FUNCTION_BLOCK PID (* Composite Function Block Type *)
  (* Standard: 61499-2 *)
  (* Version 1.0.1, 10/18/2023, ApplicationLibDevTeam, Schneider Electric, First Version *)
  PACKAGE Main;
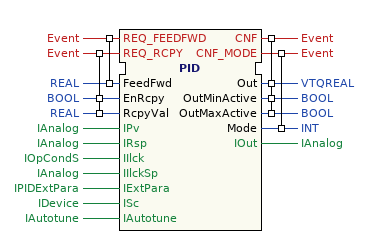
  EVENT_INPUT
    REQ_FEEDFWD WITH FeedFwd; (* Request for executing feedforward gain *)
    REQ_RCPY WITH EnRcpy, RcpyVal; (* Request for actuator position *)
  END_EVENT
  EVENT_OUTPUT
    CNF WITH Out, OutMinActive, OutMaxActive; (* Cyclic execution confirmation *)
    CNF_MODE WITH Mode; (* Execution of confirmation current setpoint *)
  END_EVENT
  VAR_INPUT
    FeedFwd : REAL; (* Feed forward value *)
    EnRcpy : BOOL; (* 1 = the RCPY is enabled *)
    RcpyVal : REAL; (* RCPY value (actuator position) *)
  END_VAR
  VAR_OUTPUT
    Out : VTQREAL; (* Calculated output value *)
    OutMinActive : BOOL; (* 1 = Out has reached OutMin Limit *)
    OutMaxActive : BOOL; (* 1 = Out has reached OutMax Limit *)
    Mode : INT; (* Current mode selected for PID calculation *)
  END_VAR
  SOCKETS
    IPv : IAnalog; (* Process value (range considered) interface adapter *)
    IRsp : IAnalog; (* Program remote setpoint interface adapter *)
    IIlck : IOpCondS; (* Interlock condition summary chain input from ilckCondItem blocks *)
    IIlckSp : IAnalog; (* Interlock setpoint interface adapter, Setpoint to be considered if interlock condition is active *)
    IExtPara : IPIDExtPara; (* External PID parameters interface adapter *)
    ISc : IDevice; (* Sequence control adapter, Controls the block when owner is in program local *)
    IAutotune : IAutotune;
  END_SOCKETS
  PLUGS
    IOut : IAnalog; (* Current output status Interface adapter *)
  END_PLUGS
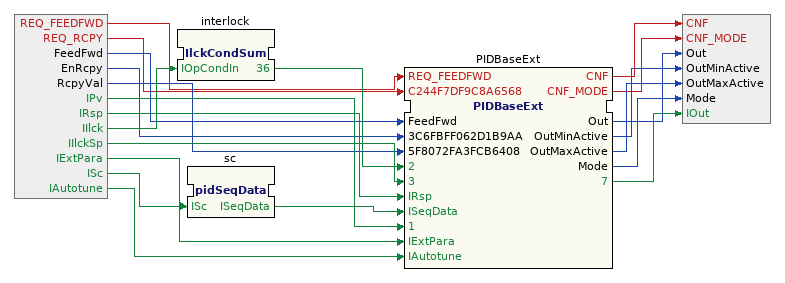
  (* PID Control *)
  (* Interlock *)
  (* Sequence Control *)
  FBS
    interlock : IlckCondSum; {SET_ATTRIBUTE(Configuration.Component.HideUnusedPorts, )}
    sc : pidSeqData;
    PIDBaseExt : PIDBaseExt;
  END_FBS
  EVENT_CONNECTIONS
    REQ_FEEDFWD TO PIDBaseExt.REQ_FEEDFWD;
    PIDBaseExt.CNF TO CNF;
    PIDBaseExt.CNF_MODE TO CNF_MODE;
    REQ_RCPY TO PIDBaseExt.C244F7DF9C8A6568;
  END_CONNECTIONS
  DATA_CONNECTIONS
    FeedFwd TO PIDBaseExt.FeedFwd;
    PIDBaseExt.Out TO Out;
    PIDBaseExt.OutMinActive TO OutMinActive;
    PIDBaseExt.OutMaxActive TO OutMaxActive;
    PIDBaseExt.Mode TO Mode;
    EnRcpy TO PIDBaseExt.3C6FBFF062D1B9AA;
    RcpyVal TO PIDBaseExt.5F8072FA3FCB6408;
  END_CONNECTIONS
  ADAPTER_CONNECTIONS
    ISc TO sc.ISc;
    IIlck TO interlock.IOpCondIn;
    interlock.36 TO PIDBaseExt.2;
    IIlckSp TO PIDBaseExt.3;
    IRsp TO PIDBaseExt.IRsp;
    sc.ISeqData TO PIDBaseExt.ISeqData;
    IPv TO PIDBaseExt.1;
    PIDBaseExt.7 TO IOut;
    IExtPara TO PIDBaseExt.IExtPara;
    IAutotune TO PIDBaseExt.IAutotune;
  END_CONNECTIONS
END_FUNCTION_BLOCK
